FUNCTION_BLOCK Q_StringValue (* Command Change String Value ( Part 6 - F.24 ) *)
  (* Standard: ISO 11783-6; Description: Copyright (c) 2022 HR Agrartechnik GmbH This program and the accompanying materials are made available under the terms of the Eclipse Public License 2.0 which is available at https://www.eclipse.org/legal/epl-2.0/ SPDX-License-Identifier: EPL-2.0 see Description Tab *)
  (* Version 1.0, 2022-07-08, Franz Höpfinger, HR Agrartechnik GmbH *)
  PACKAGE isobus::UT::Q;
  IMPORT eclipse4diac::core::TypeHash;
  IMPORT isobus::UT::Q::IDs::ID_NULL;
  (* Documentation:
  Command Change String Value with command buffer reference ( Part 6 - F.24 )
   This command sends a string to the VT. If the ObjectID is already in the command FIFO then the value of this FIFO entry is updated. The length of the string including '\0' may not be longer than the define ISO_VTC_CMD_STR_MAX_LENGTH. Take care that '\0' is trailed.
   param[in] {objectId, iso_u16}
   Object ID
   param[in] {string[], const uint8_t[] }
   Pointer to string/p> Return Values: 
   int16_t
    - VT_E_NO_ERR (0) - OK
   - VT_E_OVERFLOW (-6) - buffer overflow
   - VT_E_NOACT (-8) - Command not possible in current state
   - VT_E_NO_INSTANCE (-21) - No VT client available
   - VT_E_ISO_INSTANCE_INVALID (-129) - Identifier for instance (connection) invalid
   - VT_E_NOT_ALIVE (-130) - Identifier for instance valid, but VT Dead.
  *)
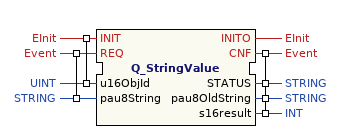
  EVENT_INPUT
    INIT : EInit WITH u16ObjId; (* Service Initialization *)
    REQ WITH pau8String; (* Service Request *)
  END_EVENT
  EVENT_OUTPUT
    INITO : EInit; (* Initialization Confirm *)
    CNF WITH STATUS, pau8OldString, s16result; (* Confirmation of Requested Service *)
  END_EVENT
  VAR_INPUT
    u16ObjId : UINT := ID_NULL; (* Object ID *)
    pau8String : STRING; (* Pointer to string *)
  END_VAR
  VAR_OUTPUT
    STATUS : STRING; (* Service Status *)
    pau8OldString : STRING; (* Old pointer to string *)
    s16result : INT; (* retval see description *)
  END_VAR
END_FUNCTION_BLOCK
